(* IEC 61131-3 sources: MSMP/PLC_Master/Source/FB, 17 files *)

(* ---- FB_AlarmManager.st ---- *)
FUNCTION_BLOCK FB_AlarmManager
VAR_INPUT Enable:BOOL; END_VAR
VAR_OUTPUT AlarmPresent:BOOL; END_VAR
AlarmPresent:=FALSE;
// TODO: Evaluate station alarms
END_FUNCTION_BLOCK

(* ---- FB_CommunicationMonitor.st ---- *)
FUNCTION_BLOCK FB_CommunicationMonitor
VAR_INPUT
 Connected:BOOL;
END_VAR
VAR_OUTPUT
 Online:BOOL;
 Alarm:BOOL;
END_VAR
Online:=Connected;
Alarm:=NOT Connected;
END_FUNCTION_BLOCK

(* ---- FB_GatewayInterface.st ---- *)
FUNCTION_BLOCK FB_GatewayInterface
VAR_INPUT
 Enable:BOOL;
END_VAR
VAR_OUTPUT
 Connected:BOOL;
END_VAR
Connected:=Enable;
// TODO: Send JSON to MQTT Gateway
END_FUNCTION_BLOCK

(* ---- FB_HMIUpdate.st ---- *)
FUNCTION_BLOCK FB_HMIUpdate
VAR_INPUT
 Enable:BOOL;
END_VAR
VAR_OUTPUT
 Updated:BOOL;
END_VAR
Updated:=Enable;
// TODO: Copy RuntimeDB values to HMI Modbus map
END_FUNCTION_BLOCK

(* ---- FB_JSONBuilder.st ---- *)
FUNCTION_BLOCK FB_JSONBuilder
VAR_INPUT
 Enable:BOOL;
END_VAR
VAR_OUTPUT
 Done:BOOL;
END_VAR
Done:=Enable;
// TODO: Serialize RuntimeDB to JSON
END_FUNCTION_BLOCK

(* ---- FB_MasterWatchdog.st ---- *)
FUNCTION_BLOCK FB_MasterWatchdog
VAR_IN_OUT Counter:DWORD;
END_VAR
Counter:=Counter+1;
END_FUNCTION_BLOCK

(* ---- FB_ModbusPolling.st ---- *)
FUNCTION_BLOCK FB_ModbusPolling
VAR_INPUT
    Enable : BOOL;
END_VAR
VAR_OUTPUT
    Busy : BOOL;
END_VAR

IF Enable THEN
    Busy := TRUE;
    // TODO: Poll all 11 Modbus RTU stations
ELSE
    Busy := FALSE;
END_IF;

END_FUNCTION_BLOCK

(* ---- FB_ModbusScheduler.st ---- *)
FUNCTION_BLOCK FB_ModbusScheduler
VAR_INPUT
 Enable:BOOL;
END_VAR
VAR_OUTPUT
 CurrentStation:INT;
 CycleComplete:BOOL;
END_VAR
VAR
 Index:INT:=1;
END_VAR

IF Enable THEN
 CurrentStation:=Index;
 Index:=Index+1;
 IF Index>11 THEN
   Index:=1;
   CycleComplete:=TRUE;
 ELSE
   CycleComplete:=FALSE;
 END_IF;
END_IF;
END_FUNCTION_BLOCK

(* ---- FB_MQTTPayload.st ---- *)
FUNCTION_BLOCK FB_MQTTPayload
VAR_INPUT
 Enable:BOOL;
END_VAR
VAR_OUTPUT
 Ready:BOOL;
END_VAR
Ready:=Enable;
// TODO: Build payload from gRuntimeDB
END_FUNCTION_BLOCK

(* ---- FB_PayloadBuilder.st ---- *)
FUNCTION_BLOCK FB_PayloadBuilder
VAR_INPUT
 Enable:BOOL;
END_VAR
VAR_OUTPUT
 Done:BOOL;
END_VAR
IF Enable THEN
 // TODO: Build payload using gRuntimeDB.Stations[1..11]
 Done:=TRUE;
ELSE
 Done:=FALSE;
END_IF;
END_FUNCTION_BLOCK

(* ---- FB_RuntimeDatabase.st ---- *)
FUNCTION_BLOCK FB_RuntimeDatabase
VAR_INPUT Enable:BOOL; END_VAR
VAR_OUTPUT Ready:BOOL; END_VAR
Ready:=Enable;
// TODO: Update Runtime Database
END_FUNCTION_BLOCK

(* ---- FB_RuntimeStatistics.st ---- *)
FUNCTION_BLOCK FB_RuntimeStatistics
VAR_OUTPUT
 OnlineStations:INT;
END_VAR
// TODO: Count online stations and update statistics
END_FUNCTION_BLOCK

(* ---- FB_RuntimeUpdate.st ---- *)
FUNCTION_BLOCK FB_RuntimeUpdate
VAR_INPUT
    Enable : BOOL;
END_VAR

IF Enable THEN
    // TODO: Copy Modbus values into Stations[]
END_IF;

END_FUNCTION_BLOCK

(* ---- FB_StationManager.st ---- *)
FUNCTION_BLOCK FB_StationManager
VAR_INPUT Enable:BOOL; END_VAR
VAR_OUTPUT Completed:BOOL; END_VAR
Completed:=Enable;
// TODO: Copy polling data into Stations[]
END_FUNCTION_BLOCK

(* ---- FB_StationPolling.st ---- *)
FUNCTION_BLOCK FB_StationPolling
VAR_INPUT
 Enable:BOOL;
END_VAR
VAR_OUTPUT
 ActiveStation:INT;
END_VAR
VAR
 i:INT;
END_VAR
IF Enable THEN
 FOR i:=1 TO 11 DO
  ActiveStation:=i;
  // TODO: Execute Modbus request for station i
 END_FOR;
END_IF;
END_FUNCTION_BLOCK

(* ---- FB_StationTimeout.st ---- *)
FUNCTION_BLOCK FB_StationTimeout
VAR_INPUT
 CommunicationOK:BOOL;
END_VAR
VAR_OUTPUT
 Timeout:BOOL;
END_VAR
Timeout:=NOT CommunicationOK;
END_FUNCTION_BLOCK

(* ---- FB_SystemStatus.st ---- *)
FUNCTION_BLOCK FB_SystemStatus
VAR_OUTPUT
 StationsOnline:INT;
END_VAR
// TODO: Count online stations
END_FUNCTION_BLOCK
